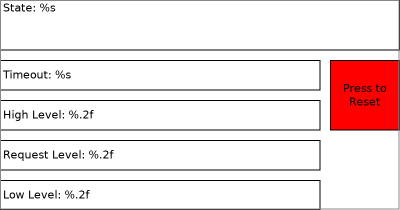
VISUALIZATION Vi_Tank  // 400x210
VAR_IN_OUT
	hmi			: Tank_Hmi;
END_VAR
    Rectangle (0,0 400x50), "State: %s", text variable: hmi.sStatusText
        p55702900: hmi.nStatusTextColor
    Rectangle (330,60 70x70), "Press to Reset", invisible if: NOT hmi.bResetButtonVis
        toggle hmi.bResetButton
    Rectangle (0,60 320x30), "Timeout: %s", text variable: Strf.SimpleTime(UDINT_TO_TIME(hmi.nTimeout.val * 1000), 'S', 'M')
        OnMouseUp: write hmi.nTimeout.val via Default, min 0
    Rectangle (0,100 320x30), "High Level: %.2f", text variable: hmi.fHighLevel.val
        OnMouseUp: write hmi.fHighLevel.val via Default, min 0
    Rectangle (0,140 320x30), "Request Level: %.2f", text variable: hmi.fRequestLevel.val
        OnMouseUp: write hmi.fRequestLevel.val via Default, min 0
    Rectangle (0,180 320x30), "Low Level: %.2f", text variable: hmi.fLowLevel.val
        OnMouseUp: write hmi.fLowLevel.val via Default, min 0
END_VISUALIZATION

(* stored: Version 1.1.0.1
   Visu Vi_Tank: Id {2685b817-12cb-488c-bf60-cfe92dc5ae11} *)
